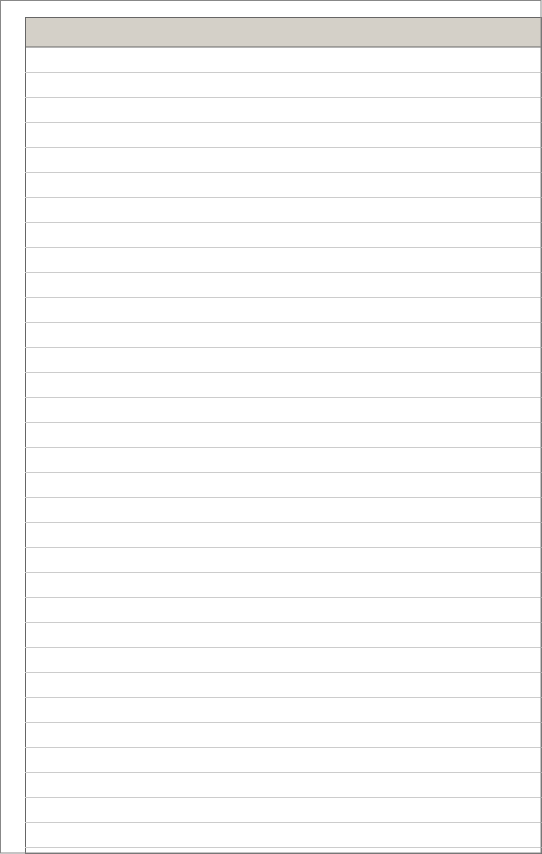
VISUALIZATION Visu_Diag  // 542x854
    Table (25,17 517x837), data array: G_Diag.aErrList
        p3854506369: G_Diag.aErrList[INDEX].horario
        p1892666644: G_Diag.aErrList[INDEX].eErrType
        p2232123230: Timestamp
        p511219082: Eror Type
END_VISUALIZATION

(* stored: Version 1.1.0.1, ProductVersion 3.1.4024.9
   Visu Visu_Diag: Id {33eaa572-2300-4ce6-8e53-b3bda5450ce4} *)
